// TwinCAT 3 PLC project reactor
// ProgramVersion: 3.1.4023.0
// libraries:
//   Tc2_Standard, * (Beckhoff Automation GmbH)
//   Tc2_System, * (Beckhoff Automation GmbH)
//   Tc3_Module, * (Beckhoff Automation GmbH)
// project tree:
//   GVLs/ GVL.TcGVL
//   / PlcTask.TcTTO
//   POUs/ MAIN.TcPOU
// real-time tasks:
//   TASK PlcTask: cycle T#10ms, priority 20, ADS port 350

CONFIGURATION reactor
    RESOURCE PLC ON TwinCAT3
        TASK PlcTask(INTERVAL := T#10ms, PRIORITY := 20);
        PROGRAM MAIN WITH PlcTask : MAIN;
    END_RESOURCE
END_CONFIGURATION

// ---- GVLs/GVL.TcGVL
{attribute 'qualified_only'}
VAR_GLOBAL
	// setpoints
	PROD_RATE					:	LREAL;	// production rate
	L_STRIPPER					:	LREAL;	// stripper level
	L_SEPARATOR					:	LREAL;	// separator level
	L_REACTOR					:	LREAL;	// reactor level
	P_REACTOR					:	LREAL;	// reactor pressure
	PCT_G_SP					:	LREAL;	// Mole percent G
	YA							: 	LREAL;	// yA 
	YAC							:	LREAL;	// yAC
	T_REACTOR					:	LREAL;	// reactor temperature
	RECYC_VALVE					:	LREAL;	// Recycle valve position
	STEAM_VALVE					:	LREAL;	// Steam valve position
	L_AGITATOR					:	LREAL;	// agitator setting		

	// actual production metrics
	COST						:	LREAL :=0.0;
	PctG						:	LREAL :=0.0;

	// process variables
	XMEAS						:	ARRAY[1..41] OF LREAL;
	XMV							:	ARRAY[1..12] OF LREAL;
	
	// shutdown indicator
	SD_FLAG						: 	BOOL	:= FALSE;

	// operating time
	OPTIME					:	LREAL := 0.0;	
	
END_VAR

// ---- POUs/MAIN.TcPOU
PROGRAM MAIN
VAR
END_VAR

END_PROGRAM
